FUNCTION_BLOCK PressureGradient
VAR_INPUT
	TotalVolume: LREAL;
	BulkModulus: LREAL;
	FlowrateIn: LREAL;
	FlowrateOut: LREAL;
	par : ST_pValveControlledCylinder;
END_VAR
VAR_OUTPUT
	PressureGradientBar : LREAL;
	PressureGradientPascal : LREAL;
	PressureBar : LREAL;
	PressurePascal : LREAL;
END_VAR
VAR
	ssMethodType : SINT := 1; 
	fbPressurePascal : DiscreteIntegrator;
END_VAR


(* Outputs for Atomic SubSystem: '<Root>/PressureGradient' *)
(* Outport: '<Root>/PressureGradientb' incorporates:
 *  Gain: '<S1>/Conv.2'
 *  Product: '<S1>/Product'
 *  Product: '<S1>/Product1'
 *  Sum: '<S1>/Sum' *)
 
//PressureGradient in [Pascal/s]
PressureGradientPascal := ((FlowrateIn - FlowrateOut)) * (par.BulkModulus / TotalVolume) * 1E5;
(* End of Outputs for SubSystem: '<Root>/PressureGradient' *)


//Pressure in [Pascal]
fbPressurePascal(
	ssMethodType := ssMethodType,
	In1 := PressureGradientPascal,
	Out1 => PressurePascal
	);

END_FUNCTION_BLOCK

(* stored: Version 1.1.0.1, ProductVersion 3.1.4024.9
   POU PressureGradient: Id {0ae25e94-6017-429e-9462-38875999b492}, SpecialFunc None *)
